FUNCTION_BLOCK EL1144
VAR
	_io : EL1xx4_Data;
	{attribute addProperty Name "WcState"}
	_wcState : WcStateInputToggle;
	{attribute addProperty Name "Info data"}
	_infoData : InfoDataBase;
END_VAR

PROPERTY IO : REFERENCE TO EL1xx4_Data
GET
IO REF= _io;
END_GET
END_PROPERTY

PROPERTY WcState : REFERENCE TO WcStateInputToggle
GET
WcState REF= _wcState;
END_GET
END_PROPERTY

END_FUNCTION_BLOCK

(* stored: Version 1.1.0.1, ProductVersion 3.1.4024.9
   POU EL1144: Id {7f90218e-7389-04bb-12db-3134105909f1}, SpecialFunc None
   Property IO: Id {0029fef6-4a93-05a3-1307-3dc36e7818ac}
   Get Get: Id {dfc01045-1c27-0188-3fde-052d5c57ba9b}
   Property WcState: Id {b6282361-c141-0bc1-168b-3e6a79633c92}
   Get Get: Id {dd93590c-2f95-01c3-35cc-19511d8c75b4} *)
